TYPE TYP_DC_MOTOR_HW :
STRUCT
	In : TYP_DC_MOTOR_HW_IN;
	Out : TYP_DC_MOTOR_HW_OUT;
END_STRUCT
END_TYPE

(* stored: Version 1.1.0.1, ProductVersion 3.1.4024.12
   DUT TYP_DC_MOTOR_HW: Id {84b65175-43a2-47b0-b978-e4315ddde008} *)
